TYPE ST_SensorData :
STRUCT
	sSensorId : STRING:='';
	rSensorValue : REAL;
END_STRUCT
END_TYPE

(* stored: Version 1.1.0.1, ProductVersion 3.1.4024.9
   DUT ST_SensorData: Id {abe01dc3-3b4c-4517-9acd-87132fce5d45} *)
